PROGRAM F95_CameraTest
VAR
	aScannerCtrl						: ARRAY[1..3] OF FB_SCANNER_CameraSelect;
	aPackScanner						: ARRAY[1..2] OF ST_SCANNER_CameraMap;

	aCameraCtrl						: ARRAY[1..2] OF FB_SCANNER_CameraSelectExt;
	aCameraEvaluation				: ARRAY[1..2] OF FB_SCANNER_Evaluation;
	
	bTemp: BOOL;
	nCameraType	: INT := 1;


	tonEnableCameraSystem: TON;
	bEnablePackAggregationCameraSystem: BOOL;
	bEnablePackTriggeringAfterDelay: BOOL;
	
	bExtract		: BOOL;
	rtExtract		: r_trig;
	
	sDataString : T_LongString;
	sDataStringTemp1 : T_LongString := '$01ST=53;$02CT=10;DS=GZDNP5JOA3IL;OG=3;XP=-50;YP=50;AP=-88;CS=06.2;SC=0070;QS=3;PN=1;$03$04$01ST=53;$02CT=10;DS=N7E1Y89UNK3O;OG=3;XP=-50;YP=-50;AP=-88;CS=06.2;SC=0070;QS=3;PN=2;$03$04DUPA'; 
	sPartitionMark	: STRING;
	nPositionMarkPos	: UINT;
	sDataField1 : T_LongString;
	
	fbExtractAnyString		: FB_ExtractAnyString;
	sDataStringTemp2 	: T_LongString := '$01ST=53;$02CT=10;DS=GZDNP5JOA3IL;OG=3;XP=-50;YP=50;AP=-88;CS=06.2;SC=0070;QS=3;PN=1;$03$04$01ST=53;$02CT=10;DS=N7E1Y89UNK3O;OG=3;XP=-50;YP=-50;AP=-88;CS=06.2;SC=0070;QS=3;PN=2;$03$04DUPA'; 
	sDataField2		: T_LongString;
	sDataField3		: T_LongString;
END_VAR

CASE nCameraType OF

1:
	CAMERA_NEWSTRUCT();
2:

	;

ELSE
;
END_CASE

//sDataString := '$01ST=53;$02CT=10;DS=GZDNP5JOA3IL;OG=3;XP=-50;YP=50;AP=-88;CS=06.2;SC=0070;QS=3;PN=1;$03$04$01ST=53;$02CT=10;DS=N7E1Y89UNK3O;OG=3;XP=-50;YP=-50;AP=-88;CS=06.2;SC=0070;QS=3;PN=2;$03$04DUPA'; 

rtExtract(CLK:=bExtract);

IF rtExtract.Q THEN
	
	//sDataStringTemp1 := sDataString;
	sPartitionMark := '$04';
	
	//nPositionMarkPos := TO_UINT(FIND2(ADR(sDataStringTemp1),ADR(sPartitionMark)));
	
	//sDataField1 := F_LongLEFT(sDataStringTemp1, TO_UINT(nPositionMarkPos)  -1); (* -1 so we don't copy the Position mark *)
	//sDataStringTemp1 := F_LongDELETE(sDataStringTemp1, nPositionMarkPos  -1 + TO_UINT(LEN(sPartitionMark)), 1);	(* Remove used data and position mark from code message string *)
	//DELETE2(ADR(sDataStringTemp1), ADR(sDataStringTemp1), SIZEOF(sDataStringTemp1), nPositionMarkPos  -1 + LEN2(ADR(sPartitionMark)), 1);
	
	//sDataStringTemp2 := sDataString;
	
	fbExtractAnyString(
	bExtractData:= TRUE, 
	nExtractChars:= 0, 
	sPrefix:= '' , 
	sSuffix:= sPartitionMark, 
	bIgnoreCase:= TRUE , 
	eExtractMode:= E_STRING_ExtrMode.WITHOUTIDENT_REMIDENT_PURGE, 
	sDataString:= sDataStringTemp2, 
	bStringFound=> , 
	sExtractedString=> sDataField2 , 
	nExtractedStringPos=> , 
	nExtractedStringLen=> , 
	nDataStringLen=> );
	
	IF NOT fbExtractAnyString.bStringFound THEN
		sDataField3 := sDataStringTemp2;
		sDataStringTemp2 := '';
		
	END_IF
END_IF

ACTION CAMERA_NEWSTRUCT:
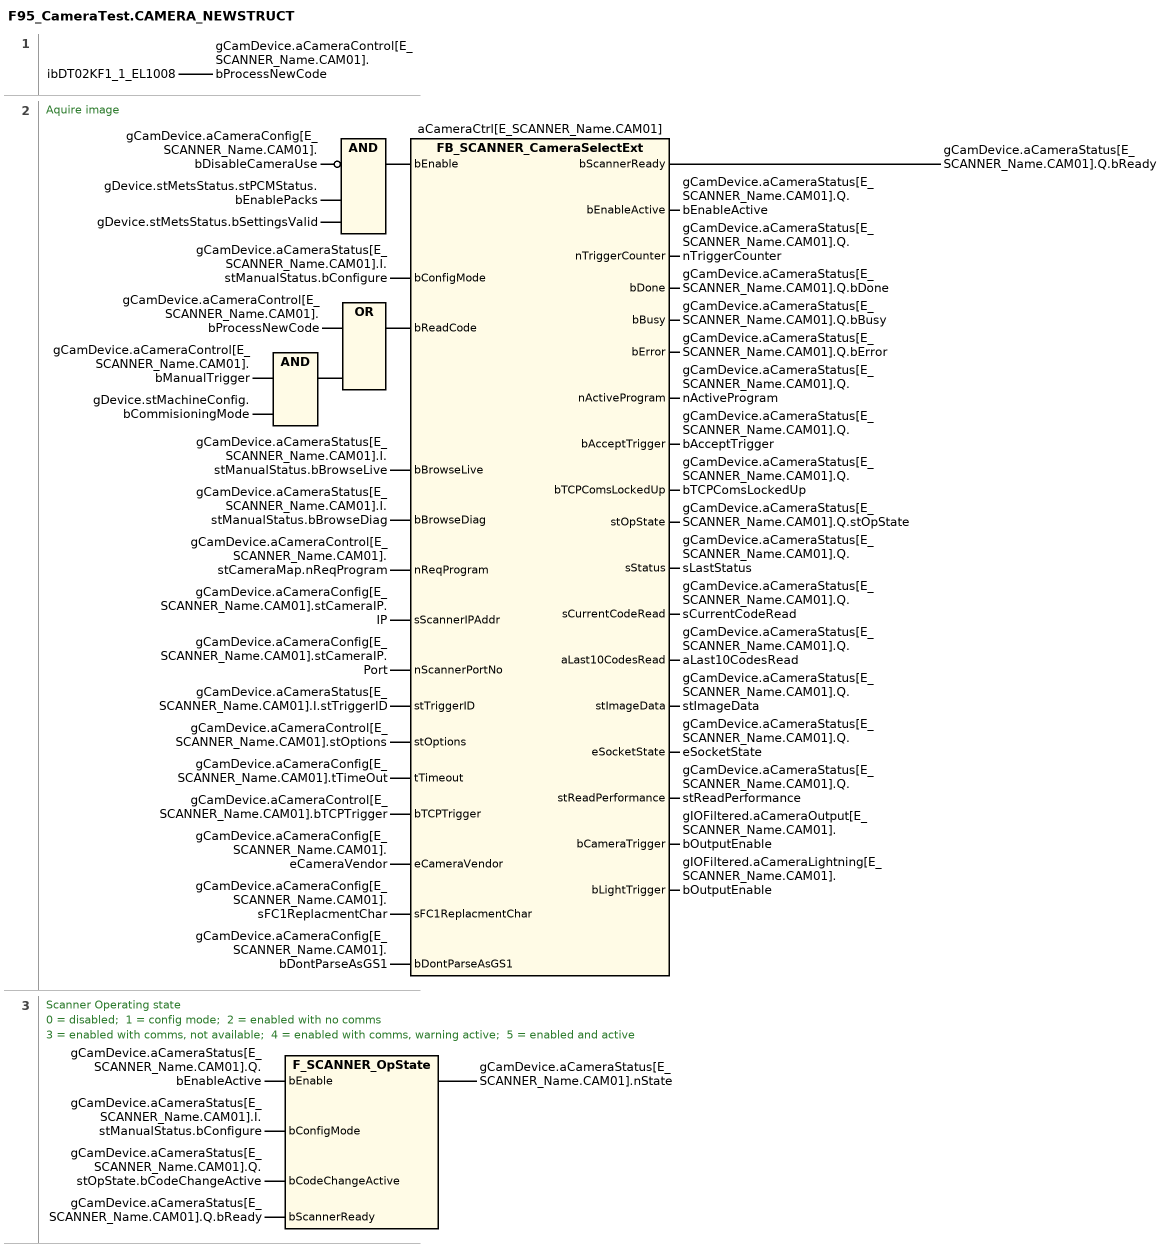
// NETWORK 1
gCamDevice.aCameraControl[E_SCANNER_Name.CAM01].bProcessNewCode := ibDT02KF1_1_EL1008;

// NETWORK 2
// Aquire image
aCameraCtrl[E_SCANNER_Name.CAM01](
    bEnable := NOT gCamDevice.aCameraConfig[E_SCANNER_Name.CAM01].bDisableCameraUse AND gDevice.stMetsStatus.stPCMStatus.bEnablePacks AND gDevice.stMetsStatus.bSettingsValid,
    bConfigMode := gCamDevice.aCameraStatus[E_SCANNER_Name.CAM01].I.stManualStatus.bConfigure,
    bReadCode := gCamDevice.aCameraControl[E_SCANNER_Name.CAM01].bProcessNewCode OR gCamDevice.aCameraControl[E_SCANNER_Name.CAM01].bManualTrigger AND gDevice.stMachineConfig.bCommisioningMode,
    bBrowseLive := gCamDevice.aCameraStatus[E_SCANNER_Name.CAM01].I.stManualStatus.bBrowseLive,
    bBrowseDiag := gCamDevice.aCameraStatus[E_SCANNER_Name.CAM01].I.stManualStatus.bBrowseDiag,
    nReqProgram := gCamDevice.aCameraControl[E_SCANNER_Name.CAM01].stCameraMap.nReqProgram,
    sScannerIPAddr := gCamDevice.aCameraConfig[E_SCANNER_Name.CAM01].stCameraIP.IP,
    nScannerPortNo := gCamDevice.aCameraConfig[E_SCANNER_Name.CAM01].stCameraIP.Port,
    stTriggerID := gCamDevice.aCameraStatus[E_SCANNER_Name.CAM01].I.stTriggerID,
    stOptions := gCamDevice.aCameraControl[E_SCANNER_Name.CAM01].stOptions,
    tTimeout := gCamDevice.aCameraConfig[E_SCANNER_Name.CAM01].tTimeOut,
    bTCPTrigger := gCamDevice.aCameraControl[E_SCANNER_Name.CAM01].bTCPTrigger,
    eCameraVendor := gCamDevice.aCameraConfig[E_SCANNER_Name.CAM01].eCameraVendor,
    sFC1ReplacmentChar := gCamDevice.aCameraConfig[E_SCANNER_Name.CAM01].sFC1ReplacmentChar,
    bDontParseAsGS1 := gCamDevice.aCameraConfig[E_SCANNER_Name.CAM01].bDontParseAsGS1,
    bEnableActive => gCamDevice.aCameraStatus[E_SCANNER_Name.CAM01].Q.bEnableActive,
    nTriggerCounter => gCamDevice.aCameraStatus[E_SCANNER_Name.CAM01].Q.nTriggerCounter,
    bDone => gCamDevice.aCameraStatus[E_SCANNER_Name.CAM01].Q.bDone,
    bBusy => gCamDevice.aCameraStatus[E_SCANNER_Name.CAM01].Q.bBusy,
    bError => gCamDevice.aCameraStatus[E_SCANNER_Name.CAM01].Q.bError,
    nActiveProgram => gCamDevice.aCameraStatus[E_SCANNER_Name.CAM01].Q.nActiveProgram,
    bAcceptTrigger => gCamDevice.aCameraStatus[E_SCANNER_Name.CAM01].Q.bAcceptTrigger,
    bTCPComsLockedUp => gCamDevice.aCameraStatus[E_SCANNER_Name.CAM01].Q.bTCPComsLockedUp,
    stOpState => gCamDevice.aCameraStatus[E_SCANNER_Name.CAM01].Q.stOpState,
    sStatus => gCamDevice.aCameraStatus[E_SCANNER_Name.CAM01].Q.sLastStatus,
    sCurrentCodeRead => gCamDevice.aCameraStatus[E_SCANNER_Name.CAM01].Q.sCurrentCodeRead,
    aLast10CodesRead => gCamDevice.aCameraStatus[E_SCANNER_Name.CAM01].Q.aLast10CodesRead,
    stImageData => gCamDevice.aCameraStatus[E_SCANNER_Name.CAM01].Q.stImageData,
    eSocketState => gCamDevice.aCameraStatus[E_SCANNER_Name.CAM01].Q.eSocketState,
    stReadPerformance => gCamDevice.aCameraStatus[E_SCANNER_Name.CAM01].Q.stReadPerformance,
    bCameraTrigger => gIOFiltered.aCameraOutput[E_SCANNER_Name.CAM01].bOutputEnable,
    bLightTrigger => gIOFiltered.aCameraLightning[E_SCANNER_Name.CAM01].bOutputEnable); // FB_SCANNER_CameraSelectExt
gCamDevice.aCameraStatus[E_SCANNER_Name.CAM01].Q.bReady := aCameraCtrl[E_SCANNER_Name.CAM01].bScannerReady;

// NETWORK 3
// 					Scanner Operating state
// 0 = disabled;  1 = config mode;  2 = enabled with no comms
// 3 = enabled with comms, not available;  4 = enabled with comms, warning active;  5 = enabled and active
//
gCamDevice.aCameraStatus[E_SCANNER_Name.CAM01].nState := F_SCANNER_OpState(bEnable := gCamDevice.aCameraStatus[E_SCANNER_Name.CAM01].Q.bEnableActive, bConfigMode := gCamDevice.aCameraStatus[E_SCANNER_Name.CAM01].I.stManualStatus.bConfigure, bCodeChangeActive := gCamDevice.aCameraStatus[E_SCANNER_Name.CAM01].Q.stOpState.bCodeChangeActive, bScannerReady := gCamDevice.aCameraStatus[E_SCANNER_Name.CAM01].Q.bReady);

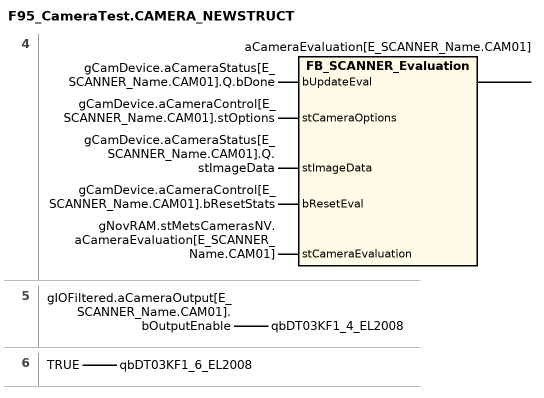
// NETWORK 4
aCameraEvaluation[E_SCANNER_Name.CAM01](
    bUpdateEval := gCamDevice.aCameraStatus[E_SCANNER_Name.CAM01].Q.bDone,
    stCameraOptions := gCamDevice.aCameraControl[E_SCANNER_Name.CAM01].stOptions,
    stImageData := gCamDevice.aCameraStatus[E_SCANNER_Name.CAM01].Q.stImageData,
    bResetEval := gCamDevice.aCameraControl[E_SCANNER_Name.CAM01].bResetStats,
    stCameraEvaluation := gNovRAM.stMetsCamerasNV.aCameraEvaluation[E_SCANNER_Name.CAM01]); // FB_SCANNER_Evaluation

// NETWORK 5
qbDT03KF1_4_EL2008 := gIOFiltered.aCameraOutput[E_SCANNER_Name.CAM01].bOutputEnable;

// NETWORK 6
qbDT03KF1_6_EL2008 := TRUE;
END_ACTION

END_PROGRAM

(* stored: Version 1.1.0.1
   POU F95_CameraTest: Id {2731e840-bfa2-45b6-baaa-9088a04fe0de}, SpecialFunc None
   Action CAMERA_NEWSTRUCT: Id {a18962f1-ca19-4d4b-b5a4-6ef06ba10dd4} *)
